Fanuc KAREL source: kt00585.KL

PROGRAM KT00585
%STACKSIZE=65535
%PRIORITY=65535
%NOLOCKGROUP
VAR
I1 : INTEGER
V2 : VECTOR
OUT : VECTOR
BEGIN
I1=2
V2.Y=2.0
-- UNRESOLVED_PC line 10 opcodes [21 49 8B 4A] marker_code=36
END KT00585
